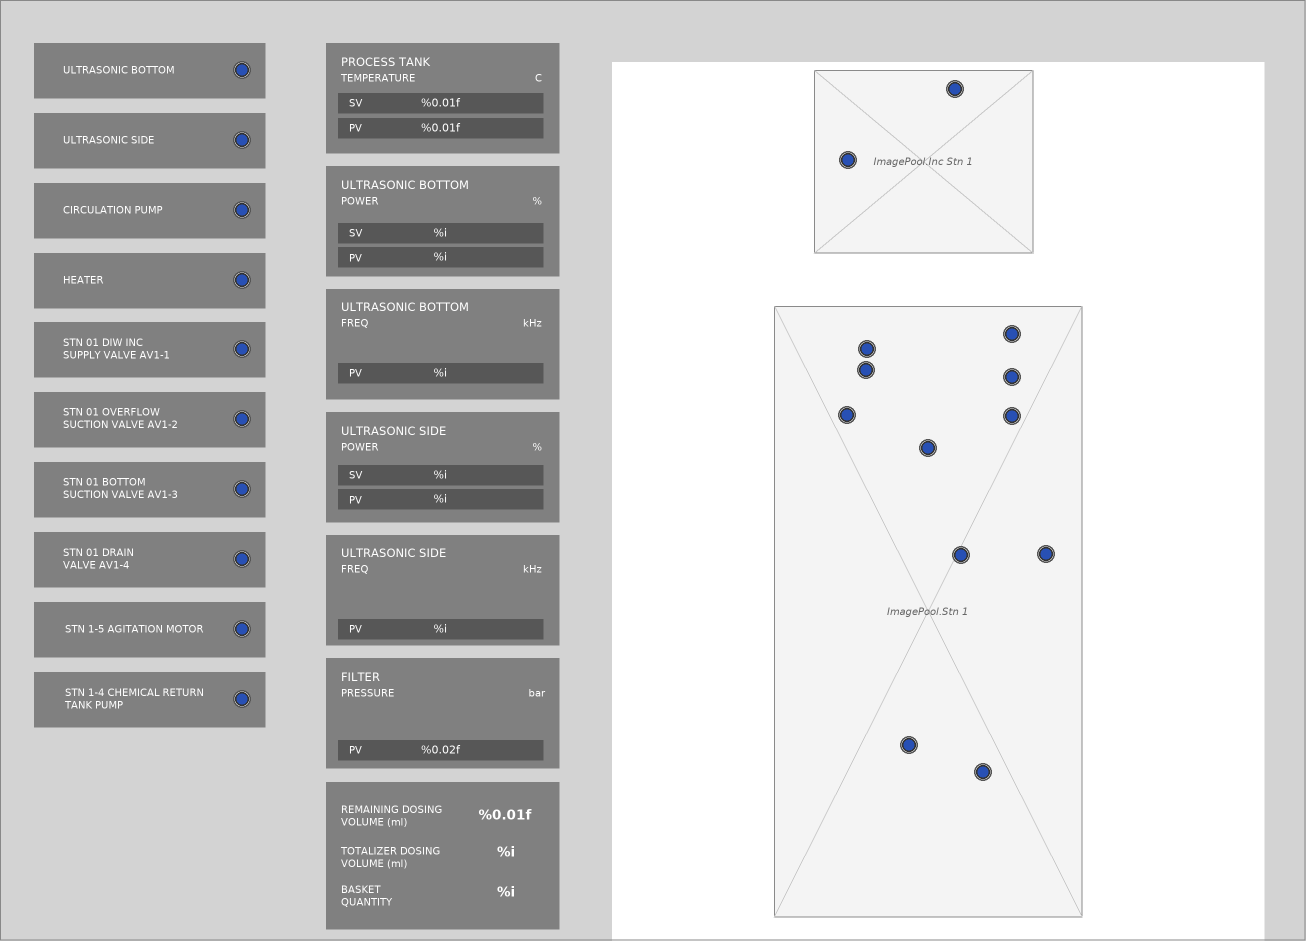
VISUALIZATION Auto_Station01  // 1306x941
    Rectangle (0,0 1306x875)
    RoundedRectangle (34,43 231x55)
    Label (60,62 163x16), "ULTRASONIC BOTTOM"
    Lamp1 (232,60 20x20), variable: ARdsMAP_HmiVariableStn[1].bProTankUsBtm_IND, style: Lamp-Lamp1-Blue
    RoundedRectangle (34,183 231x55)
    Label (60,202 151x16), "CIRCULATION PUMP"
    Lamp1 (232,200 20x20), variable: ARdsMAP_HmiVariableStn[1].bProTankPump_IND, style: Lamp-Lamp1-Blue
    RoundedRectangle (34,253 231x55)
    Label (60,272 151x16), "HEATER"
    Lamp1 (232,270 20x20), variable: ARdsMAP_HmiVariableStn[1].bProTankHeater_IND, style: Lamp-Lamp1-Blue
    RoundedRectangle (326,43 233x110)
    Label (338,54 150x16), "PROCESS TANK"
    Label (338,67 99x22), "TEMPERATURE"
    Label (516,67 29x22), "C"
    Rectangle (338,93 205x20), "%0.01f", text variable: ARrStnTempSV[1]
    Label (346,92 22x22), "SV"
    Rectangle (338,118 205x20), "%0.01f", text variable: ARrStnTempPV[1]
    Label (346,117 22x22), "PV"
    RoundedRectangle (326,166 233x110)
    Label (338,177 150x16), "ULTRASONIC BOTTOM"
    Label (338,190 99x22), "POWER"
    Label (516,190 29x22), "%"
    Rectangle (338,223 205x20), "%i", text variable: DSWeberEnclosure[1].DSWeberGenerator[2].IN_iTargetPowerPercentSetPoint
    Label (346,222 22x22), "SV"
    Rectangle (338,247 205x20), "%i", text variable: ARiStnUSBtmAPv[1]
    Label (346,247 22x22), "PV"
    Group (326,658 233x110)
        RoundedRectangle (0,0 233x110)
        Label (12,11 150x16), "FILTER"
        Label (12,24 99x22), "PRESSURE"
        Label (190,24 32x22), "bar"
        Rectangle (12,82 205x20), "%0.02f", text variable: ARrStnFilterPressurePV[1]
        Label (20,81 22x22), "PV"
    Group (326,289 233x110)
        RoundedRectangle (0,0 233x110)
        Label (12,23 99x22), "FREQ"
        Label (12,10 150x16), "ULTRASONIC BOTTOM"
        Label (190,23 29x22), "kHz"
        Rectangle (12,74 205x20), "%i", text variable: ARiStnUSBtmAFreqPv[1]
        Label (20,73 22x22), "PV"
    RoundedRectangle (34,322 231x55)
    Label (60,325 151x48), "STN 01 DIW INC SUPPLY VALVE AV1-1"
    Lamp1 (232,339 20x20), variable: ARdsMAP_HmiVariableStn[1].bValve01_IND, style: Lamp-Lamp1-Blue
    RoundedRectangle (34,602 231x55)
    Label (62,611 160x36), "STN 1-5 AGITATION MOTOR"
    Lamp1 (232,619 20x20), variable: ARdsMAP_HmiVariableGeneral.bProTankAgitationMotor_IND, style: Lamp-Lamp1-Blue
    RoundedRectangle (34,392 231x55)
    Lamp1 (232,409 20x20), variable: ARdsMAP_HmiVariableStn[1].bValve02_IND, style: Lamp-Lamp1-Blue
    Label (60,394 168x49), "STN 01 OVERFLOW SUCTION VALVE AV1-2"
    RoundedRectangle (326,782 233x147)
    Label (338,840 118x35), "TOTALIZER DOSING VOLUME (ml)"
    Label (338,802 118x28), "REMAINING DOSING VOLUME (ml)"
    Rectangle (464,801 82x28), "%0.01f", text variable: ARDSProminentDosingHMI[1].Out_rRemainedDosingVolume_ml
    Rectangle (465,838 82x28), "%i", text variable: ARDSProminentDosingHMI[1].Out_iDosingTotalizer_ml
    Label (338,882 118x28), "BASKET QUANTITY"
    Rectangle (465,878 82x28), "%i", text variable: ARDSProminentDosingHMI[1].Out_iBasketQtyBeforeAutoDosingPV
    RoundedRectangle (34,113 231x55)
    Label (60,132 163x16), "ULTRASONIC SIDE"
    Lamp1 (232,130 20x20), variable: ARdsMAP_HmiVariableStn[1].bProTankUsSide_IND, style: Lamp-Lamp1-Blue
    RoundedRectangle (34,462 231x55)
    Label (60,465 151x47), "STN 01 BOTTOM SUCTION VALVE AV1-3"
    Lamp1 (232,479 20x20), variable: ARdsMAP_HmiVariableStn[1].bValve03_IND, style: Lamp-Lamp1-Blue
    RoundedRectangle (34,532 231x55)
    Lamp1 (232,549 20x20), variable: ARdsMAP_HmiVariableStn[1].bValve04_IND, style: Lamp-Lamp1-Blue
    Label (60,536 168x46), "STN 01 DRAIN VALVE AV1-4"
    RoundedRectangle (34,672 231x55)
    Label (62,674 170x50), "STN 1-4 CHEMICAL RETURN TANK PUMP"
    Lamp1 (232,689 20x20), variable: ARdsMAP_HmiVariableGeneral.bProTankPump_IND, style: Lamp-Lamp1-Blue
    Group (326,412 233x110)
        RoundedRectangle (0,0 233x110)
        Label (12,11 150x16), "ULTRASONIC SIDE"
        Label (12,24 99x22), "POWER"
        Label (190,24 29x22), "%"
        Rectangle (12,53 205x20), "%i", text variable: DSWeberEnclosure[1].DSWeberGenerator[1].IN_iTargetPowerPercentSetPoint
        Label (20,52 22x22), "SV"
        Rectangle (12,77 205x20), "%i", text variable: ARiStnUSSideAPv[1]
        Label (20,77 22x22), "PV"
    Group (326,535 233x110)
        RoundedRectangle (0,0 233x110)
        Label (12,23 99x22), "FREQ"
        Label (12,10 150x16), "ULTRASONIC SIDE"
        Label (190,23 29x22), "kHz"
        Rectangle (12,84 205x20), "%i", text variable: ARiStnUSSideAFreqPv[1]
        Label (20,83 22x22), "PV"
    Rectangle (612,62 652x879)
    Image (774,306 308x611), image: ImagePool.Stn 1
    Lamp1 (918,438 20x20), variable: ARdsMAP_HmiVariableStn[1].bProTankUsBtm_IND, style: Lamp-Lamp1-Blue
    Lamp1 (899,735 20x20), variable: ARdsMAP_HmiVariableStn[1].bProTankPump_IND, style: Lamp-Lamp1-Blue
    Lamp1 (856,360 20x20), variable: ARdsMAP_HmiVariableStn[1].bProTankHeater_IND, style: Lamp-Lamp1-Blue
    Lamp1 (1036,544 20x20), variable: ARdsMAP_HmiVariableStn[1].bValve02_IND, style: Lamp-Lamp1-Blue
    Lamp1 (837,405 20x20), variable: ARdsMAP_HmiVariableStn[1].bProTankUsSide_IND, style: Lamp-Lamp1-Blue
    Lamp1 (951,545 20x20), variable: ARdsMAP_HmiVariableStn[1].bValve03_IND, style: Lamp-Lamp1-Blue
    Lamp1 (973,762 20x20), variable: ARdsMAP_HmiVariableStn[1].bValve04_IND, style: Lamp-Lamp1-Blue
    Lamp1 (857,339 20x20), variable: ARdsMAP_HmiVariableStn[1].bProcessTankMinLevel_IND, style: Lamp-Lamp1-Blue
    Lamp1 (1002,324 20x20), variable: ARdsMAP_HmiVariableStn[1].bOverflowMaxLevel_IND, style: Lamp-Lamp1-Blue
    Lamp1 (1002,367 20x20), variable: ARdsMAP_HmiVariableStn[1].bOverflowMinLevel_IND, style: Lamp-Lamp1-Blue
    Lamp1 (1002,406 20x20), variable: ARdsMAP_HmiVariableStn[1].bProTankUsSide_IND, style: Lamp-Lamp1-Blue
    Image (814,70 219x183), image: ImagePool.Inc Stn 1
    Lamp1 (945,79 20x20), variable: ARdsMAP_HmiVariableStn[1].bValve01_IND, style: Lamp-Lamp1-Blue
    Lamp1 (838,150 20x20), variable: ARdsMAP_HmiVariableStn[1].bDosingPump_IND, style: Lamp-Lamp1-Blue
END_VISUALIZATION

(* stored: Version 1.1.0.1, ProductVersion 3.1.4024.12
   Visu Auto_Station01: Id {4e780cb0-6ca2-421d-be85-7db6f61f1a1f} *)
